(* IEC 61131-3 sources: Industry-PLC-LLM/data/PLCBEAD_repo/PLCBEAD_PLCEmbed-main/PLC-BEAD/Source/GEB/ISC_NUM, 1 file *)

(* ---- ISC_NUM.ST ---- *)
FUNCTION ISC_NUM:BOOL

	VAR_INPUT
		IN :	BYTE;
	END_VAR

	ISC_NUM := IN > BYTE#47 AND IN < BYTE#58;

END_FUNCTION

PROGRAM program0
	VAR
		IN : BYTE;
		OUT : BOOL;
	END_VAR

	OUT := ISC_NUM(IN);
END_PROGRAM
